Universal Robots PolyScope program: universal_robots_robot_motion_script.urp

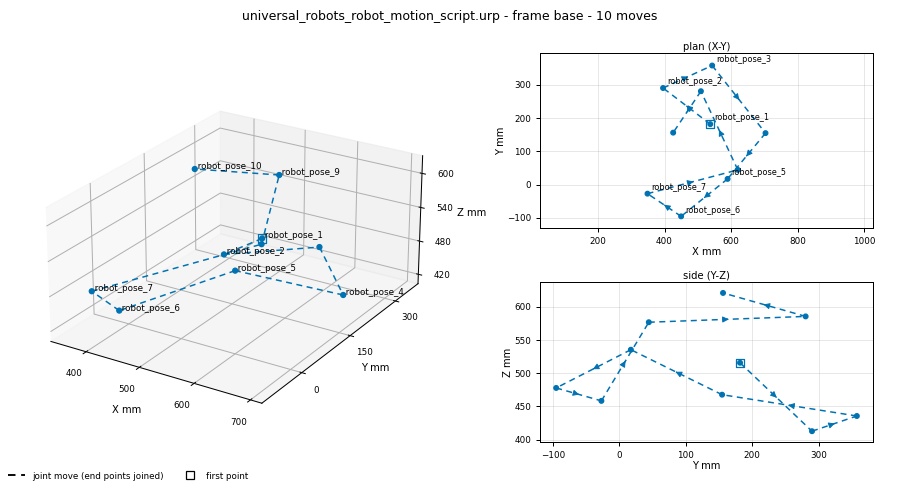
[picture p0: tool path of universal_robots_robot_motion_script.urp in frame base, 10 of 10 moves have a stored position in this frame; points joined in program order, loops and branches not executed]
Program hand_eye_script (installation=calibboard directory=/programs/usbdisk createdIn=5.5.1.82186 lastSavedIn=5.5.1.82186 robotSerialNumber=20195501515)
Calibrated DH parameters: a=[0.000072, -0.399805, -0.37789, 0.000062, -0.000013, 0]; d=[0.162483, 48.810299, -65.8047, 17.127566, 0.099809, 0.099443]; alpha=[1.570513, -0.002952, 0.006175, 1.570711, -1.57004, 0]; deltaTheta=[0, -0.345938, 0.075062, 0.270887, -0.000041, 0]
InitVariablesNode variables(variable(name=Counter, expression=0))
Robot Program (runOnlyOnce=false)
  'set image_counter to 0'
  Script: write_output_integer_register(24,0)
  'set start_capture to False'
  Script: write_output_boolean_register(64,False)
  SuppressedNode
    Wait DigitalInput pin=GP_bool_in[65]; digitalValue=1
  Wait Condition expression=read_input_boolean_register(65)
  Script: read_input_boolean_register(65)
  'Add, alter, or remove waypoints to calibrate'
  MoveJ speed 15 deg/s, acceleration 15 deg/s^2 (useActiveTCP=true) feature=Base
    Waypoint robot_pose_1: TCP in base x=537.26 y=181.734 z=515.774 mm, rx=-3.103 ry=-0.0398 rz=-0.0836 rad; joints [32.056, -97.252, -79.274, -89.771, 90.491, -59.17] deg; TCP offset x=0 y=0 z=0 mm, rx=0 ry=0 rz=0 rad
    Call capture_hand_eye
    Waypoint robot_pose_2: TCP in base x=395.585 y=290.198 z=412.678 mm, rx=2.8016 ry=0.2926 rz=0.5243 rad; joints [57.196, -86.477, -106.266, -76.71, 63.973, -44.519] deg
    Call capture_hand_eye
    Waypoint robot_pose_3: TCP in base x=542.989 y=357.749 z=435.584 mm, rx=2.5453 ry=0.9249 rz=-0.3097 rad; joints [47.399, -115.669, -61.851, -115.488, 75.431, -79.411] deg
    Call capture_hand_eye
    Waypoint robot_pose_4: TCP in base x=703.239 y=154.713 z=467.688 mm, rx=-3.011 ry=-0.0228 rz=0.4774 rad; joints [21.432, -127.267, -39.977, -117.888, 101.559, -70.906] deg
    Call capture_hand_eye
    Waypoint robot_pose_5: TCP in base x=589.371 y=17.263 z=535.466 mm, rx=-2.3215 ry=-1.7258 rz=0.1061 rad; joints [12.688, -105.199, -63.752, -110.757, 101.485, -151.413] deg
    Call capture_hand_eye
    Waypoint robot_pose_6: TCP in base x=449.771 y=-95.295 z=477.854 mm, rx=-2.7153 ry=-0.6585 rz=-0.2662 rad; joints [0.003, -83.033, -100.778, -79.878, 111.46, -115.776] deg
    Call capture_hand_eye
    Waypoint robot_pose_7: TCP in base x=348.761 y=-27.134 z=458.385 mm, rx=-2.5599 ry=-1.7373 rz=-0.4822 rad; joints [15.718, -63.745, -119.19, -70.39, 96.365, -141.348] deg
    Call capture_hand_eye
    Waypoint robot_pose_8: TCP in base x=620.061 y=44.293 z=576.873 mm, rx=-2.9184 ry=0.3268 rz=0.2327 rad; joints [14.148, -110.142, -52.18, -112.309, 103.943, -63.544] deg
    Call capture_hand_eye
    Waypoint robot_pose_9: TCP in base x=509.17 y=280.611 z=585.647 mm, rx=2.8969 ry=-0.0142 rz=0.0471 rad; joints [43.964, -104.154, -57.76, -116.693, 79.015, -44.544] deg
    Call capture_hand_eye
    Waypoint robot_pose_10: TCP in base x=425.873 y=156.132 z=621.007 mm, rx=3.0868 ry=0.0606 rz=0.3616 rad; joints [39.213, -81.821, -80.746, -98.079, 80.614, -53.624] deg
    Call capture_hand_eye
  'Calibration complete'
  SuppressedNode
    Set ExpressionOutput pin=GP_int_out[24]; expression=-1
  Script: write_output_integer_register(24,-1)
  Halt
SubProgram -> capture_hand_eye
SubProgram capture_hand_eye (keepSynchronizedWithDisk=false)
  Wait Sleep waitTime=2
  Counter := Counter+1
  SuppressedNode
    Set ExpressionOutput pin=GP_int_out[24]; expression=Counter
  Script: write_output_integer_register(24,Counter)
  SuppressedNode
    Set DigitalOutput pin=GP_bool_out[64]; digitalValue=1
  Script: write_output_boolean_register(64, True)
  Wait Condition expression=read_input_boolean_register(64)
  SuppressedNode
    Set DigitalOutput pin=GP_bool_out[64]; digitalValue=0
  Script: write_output_boolean_register(64, False)
